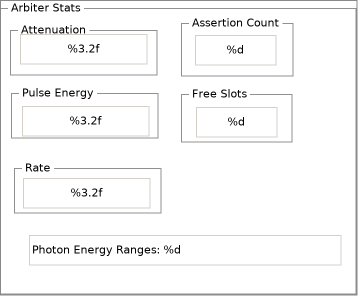
VISUALIZATION ArbiterStats  // 358x296
VAR_IN_OUT
	fbArbiter	:	FB_Arbiter;
END_VAR
    GroupBox (0,0 356x294), "Arbiter Stats"
        GroupBox (10,22 147x53), "Attenuation"
            Textfield (10,12 127x30), "%3.2f", text variable: fbArbiter.q_stBeamParams.fAtt
        GroupBox (11,85 147x53), "Pulse Energy"
            Textfield (11,21 127x30), "%3.2f", text variable: fbArbiter.q_stBeamParams.fPP_mJ
        GroupBox (14,160 147x53), "Rate"
            Textfield (9,18 127x30), "%3.2f", text variable: fbArbiter.stOutputBP.nRate
        GroupBox (181,15 112x61), "Assertion Count"
            Textfield (14,20 81x30), "%d", text variable: fbArbiter.fbBPAssertionPool.hTable.nCount
        GroupBox (181,86 111x56), "Free Slots"
            Textfield (15,21 81x30), "%d", text variable: fbArbiter.fbBPAssertionPool.hTable.nFree
        Textfield (29,235 312x30), "Photon Energy Ranges: %d", text variable: fbArbiter.q_stBeamParams.neVRange
END_VISUALIZATION

(* stored: Version 1.1.0.1, ProductVersion 3.1.4024.0
   Visu ArbiterStats: Id {ef270ad9-bed8-084d-3237-50f5c5a698e2} *)
